/// machine data that is used through most sequences of the unit (motor speed, axes positions, ...)
TYPE AssemblyDataMachine :
STRUCT
  Slowspeed : LREAL;
  Highspeed : LREAL;
END_STRUCT
END_TYPE

(* stored: Version 1.1.0.1
   DUT AssemblyDataMachine: Id {76407625-6c44-439a-8101-e5047a3ecb0a} *)
